TYPE RendererTestStruct :
STRUCT
	_wrapLayoutTests: WrapLayoutTest;
END_STRUCT
END_TYPE

(* stored: Version 1.1.0.1, ProductVersion 3.1.4024.9
   DUT RendererTestStruct: Id {f29f5fcd-3df5-4eea-8c31-6186e4f5ace9} *)
